FUNCTION_BLOCK PUBLIC FB_LogToDisk // Regularly writes contents of the log to disk
// Once the log file reaches a set size, a new log file is created.
// If the max number of files is reached, the oldest file is discarded.
VAR CONSTANT
	MAX_ITEMS_IN_BUFFER : UDINT := 20; // Should be long enough to allow for worst case writes (where an old file has to be deleted and a new file created).  
	CRLF : STRING := '$R$L'; // Windows style line ending
END_VAR
VAR_INPUT
	bEnable : BOOL; // If enabled, log items will be written to disk
END_VAR
VAR_OUTPUT
	bFault 				: BOOL; // An error occured while trying to add to log or write to disk
	sFaultDescription	: STRING[80]; // Detailed error information
	bLoggerInitialized  : BOOL; // True the first time the logger has ran through all states (ie., after succesfully writing the first log message and emptying the buffer)
	sCurrentLogFile		: T_MaxString; // The file which is currently used for logging (and can be viewed for instance by the HMI)
END_VAR
VAR
	// Properties set by FB_init
	sLogFolder 			: T_MaxString;
	sLogFilePrefix 		: T_MaxString;
	sLogFileExtension 	: T_MaxString;
	nMaxLogFileSize 	: ULINT; // [bytes] When this size is reached, a new log file is created 
	nMaxNumberOfLogFiles: UINT;

	// State machine
	fbStateMachine 	: FB_StateMachine;	
	eState 			: E_LogToDiskState := E_LogToDiskState.InitializeFBs;
	
	// Log item buffer
	stLogItemFromBuffer : UDT_LogItem; // Log item retrieved from the buffer	
	stLogItemToDisk		: UDT_LogItem; // Log item to be written to the log file
	cbBuffer 	: ARRAY[1..(MAX_ITEMS_IN_BUFFER * (SIZEOF(UDT_LogItem) + 4))] OF BYTE; // Note that the buffer size is larger than the number of items * item size, because 4 bytes are added to each item by FB_MemRingBuffer
	fbBuffer 	: FB_MemRingBuffer := (pBuffer:= ADR(cbBuffer), cbBuffer:= SIZEOF(cbBuffer));

	// File function blocks (asynchronous)
	fbFileOpen			: FB_FileOpen; // https://infosys.beckhoff.com/content/1033/tcplclib_tc2_system/30977547.html
	fbFilePuts			: FB_FilePuts; // https://infosys.beckhoff.com/content/1033/tcplclib_tc2_system/30979083.html
	fbFileClose			: FB_FileClose; // https://infosys.beckhoff.com/content/1033/tcplclib_tc2_system/30972939.html
	fbFileProperties	: FB_FileProperties; // https://infosys.beckhoff.com/content/1033/tcplclib_tc2_utilities/10047843595.html
    fbEnumFiles			: FB_EnumFindFileEntry; // https://infosys.beckhoff.com/content/1033/tcplclib_tc2_utilities/34982539.html
	fbFileDelete		: FB_FileDelete; // https://infosys.beckhoff.com/content/1033/tcplclib_tc2_system/30974475.html

	sPath: STRING; // Path to the current log file
	
	tOldestLogFile 	: ST_FindFileEntry; // Reference to the oldest log file in the log folder
	nFileCount		: UINT; // Number of log files found  
	
	fbFormatString : FB_FormatString; // https://infosys.beckhoff.com/content/1033/tcplclib_tc2_utilities/34990219.html
END_VAR
VAR_TEMP
	fMonth : REAL;
	fDay : REAL;
	fHour : REAL;
	fMinute : REAL;
	fSecond : REAL;
	fMilliseconds : REAL;
	sLevel : T_MaxString;

	nFileSize : ULINT;
	
	stEmptyLogItem : UDT_LogItem;
END_VAR

fbStateMachine(nState := eState);

CASE eState OF
	E_LogToDiskState.InitializeFBs:
		// Initialize function blocks
		fbFileOpen(
			bExecute := FALSE,
			ePath := PATH_GENERIC,
		);
		fbFilePuts(bExecute := FALSE);
		fbFileClose(bExecute := FALSE);
		fbFileProperties(bExecute := FALSE);
		fbEnumFiles(bExecute := FALSE);
		fbFileDelete(
			bExecute := FALSE,
			ePath := PATH_GENERIC,
		);
		
		eState := E_LogToDiskState.WaitForCommand;

	E_LogToDiskState.WaitForCommand:
		IF bEnable THEN
			IF (stLogItemFromBuffer.sMsg = '') THEN
				stLogItemFromBuffer := Pop();
			ELSE
				eState := E_LogToDiskState.OpenOrCreateFile;
			END_IF
		END_IF

	E_LogToDiskState.OpenOrCreateFile:
		IF fbStateMachine.bStateChanged THEN
			// Create a new file path if none was given (i.e., after reboot or when file size limit has been reached)
			IF (sPath = '') THEN
				sPath := CreatePath();
			END_IF  	
		END_IF
		fbFileOpen(
			bExecute := TRUE,	
			sPathName := sPath, 
			nMode := FOPEN_MODEAPPEND OR FOPEN_MODETEXT, // Open file in read/write text mode
		);
		IF (NOT fbFileOpen.bBusy) THEN
			fbFileOpen(bExecute := FALSE);
			IF fbFileOpen.bError THEN
				fbFormatString(sFormat := 'Unable to open file (error code 0x%X)', arg1 := F_UDINT(fbFileOpen.nErrId), sOut => sFaultDescription);
				eState := E_LogToDiskState.Error;
			ELSE
				sCurrentLogFile := sPath;
				eState := E_LogToDiskState.CheckFileSize;
			END_IF
		END_IF

	E_LogToDiskState.CheckFileSize:
		fbFileProperties(
			bExecute := TRUE,	
			sPathName := sPath 
		);
		IF (NOT fbFileProperties.bBusy) THEN
			fbFileProperties(bExecute := FALSE);
			IF fbFileProperties.bError THEN
				fbFormatString(sFormat := 'Unable to get file properties (error code 0x%X)', arg1 := F_UDINT(fbFileProperties.nErrId), sOut => sFaultDescription);
				eState := E_LogToDiskState.Error;
			ELSE
				// Check file size
				// ST_FindFileEntry info at https://infosys.beckhoff.com/content/1033/tcplclib_tc2_utilities/35363851.html
				nFileSize := ULARGE_TO_ULINT(fbFileProperties.stProperties.fileSize);
				IF (nFileSize >= nMaxLogFileSize) THEN
					// Create a final log item for this log file
					stLogItemToDisk.eLevel := E_LogLevel.DEBUG;
					fbFormatString(
						sFormat := 'File size exceeded (%u/%u bytes), creating new file.',
						arg1 := F_ULINT(nFileSize),
						arg2 := F_ULINT(nMaxLogFileSize),
						sOut => stLogItemToDisk.sMsg
					);
					stLogItemToDisk.stTimestamp := Sys_Variables.SystemTime_TS;
					sPath := ''; // Trigger new file creation
				ELSE
					stLogItemToDisk := stLogItemFromBuffer; // Set log item to be written to disk
					stLogItemFromBuffer := stEmptyLogItem; // Clear log item from buffer to trigger new item pop
				END_IF
				eState := E_LogToDiskState.WriteLogItemPrefix;
			END_IF
		END_IF
	
	E_LogToDiskState.WriteLogItemPrefix:
		IF fbStateMachine.bStateChanged THEN
			// Build a prefix string, e.g. '[2022-02-04 12:13:45.343] INFO; '

			// Suppress error "VAR_IN_OUT parameter 'in' needs variable with write access as input."	
			fMonth := WORD_TO_REAL(stLogItemToDisk.stTimestamp.wMonth); 
			fDay := WORD_TO_REAL(stLogItemToDisk.stTimestamp.wDay); 
			fHour := WORD_TO_REAL(stLogItemToDisk.stTimestamp.wHour); 
			fMinute := WORD_TO_REAL(stLogItemToDisk.stTimestamp.wMinute); 
			fSecond := WORD_TO_REAL(stLogItemToDisk.stTimestamp.wSecond); 
			fMilliseconds := WORD_TO_REAL(stLogItemToDisk.stTimestamp.wMilliseconds);
			sLevel := TO_STRING(stLogItemToDisk.eLevel);
 
			fbFormatString(
				sFormat := '[%u-%02.0f-%02.0f %02.0f:%02.0f:%02.0f.%03.0f] %s: ',
				arg1 := F_WORD(stLogItemToDisk.stTimestamp.wYear),
				arg2 := F_REAL(fMonth),
				arg3 := F_REAL(fDay),
				arg4 := F_REAL(fHour),
				arg5 := F_REAL(fMinute),
				arg6 := F_REAL(fSecond),
				arg7 := F_REAL(fMilliseconds),
				arg8 := F_STRING(sLevel),
				sOut => fbFilePuts.sLine
			);
		END_IF
		fbFilePuts(bExecute := TRUE, hFile := fbFileOpen.hFile);
		IF (NOT fbFilePuts.bBusy) THEN
			fbFilePuts(bExecute := FALSE);
			IF fbFilePuts.bError THEN
				fbFormatString(sFormat := 'Unable to write log record to file (error code 0x%X)', arg1 := F_UDINT(fbFilePuts.nErrId), sOut => sFaultDescription);
				eState := E_LogToDiskState.Error;
			ELSE // Done, write the log message
				eState := E_LogToDiskState.WriteLogItemMessage;
			END_IF
		END_IF
	
	E_LogToDiskState.WriteLogItemMessage:
		IF fbStateMachine.bStateChanged THEN
			fbFilePuts.sLine := CONCAT(stLogItemToDisk.sMsg, CRLF); 	
		END_IF
		fbFilePuts(bExecute := TRUE, hFile := fbFileOpen.hFile);
		IF (NOT fbFilePuts.bBusy) THEN
			fbFilePuts(bExecute := FALSE);
			IF fbFilePuts.bError THEN
				fbFormatString(sFormat := 'Unable to write log record to file (error code 0x%X)', arg1 := F_UDINT(fbFilePuts.nErrId), sOut => sFaultDescription);
				eState := E_LogToDiskState.Error;
			ELSE // Done, get the next log item in the buffer
				IF (stLogItemFromBuffer.sMsg <> '') THEN 
					// Last log item retrieved from the buffer wasn't written yet (e.g., after new file creation), so no need to pop items from the buffer yet
					eState := E_LogToDiskState.CloseFile;
				ELSE // Check if there are more items in the buffer
					stLogItemFromBuffer := Pop();
					IF (stLogItemFromBuffer.sMsg = '') THEN // Buffer empty, close the file
						eState := E_LogToDiskState.CloseFile;
					ELSE // More items to be written, but first check file size before adding more items
						eState := E_LogToDiskState.CheckFileSize;
					END_IF
				END_IF
			END_IF
		END_IF
	
	E_LogToDiskState.CloseFile:
		fbFileClose(bExecute := TRUE, hFile := fbFileOpen.hFile);
		IF (NOT fbFileClose.bBusy) THEN
			fbFileClose(bExecute := FALSE);
			IF fbFileClose.bError THEN
				fbFormatString(sFormat := 'Unable to close file (error code 0x%X)', arg1 := F_UDINT(fbFileClose.nErrId), sOut => sFaultDescription);
				eState := E_LogToDiskState.Error;
			ELSE
				eState := E_LogToDiskState.FindObsoleteFiles;
			END_IF
		END_IF
	
	E_LogToDiskState.FindObsoleteFiles:
		// Delete oldest log files in log folder until we're at MAX_NUMBER_OF_LOG_FILES
		IF fbStateMachine.bStateChanged THEN
			nFileCount := 0;	
			tOldestLogFile.sFileName := ''; 
			// Create a path search string, e.g. '/tmp/Log_*.txt'
			fbFormatString(
				sFormat := '%s/%s*.%s',
				arg1 := F_STRING(sLogFolder),
				arg2 := F_STRING(sLogFilePrefix),
				arg3 := F_STRING(sLogFileExtension),
				sOut => fbEnumFiles.sPathName
			);
			fbEnumFiles.eCmd := E_EnumCmdType.eEnumCmd_First;
		END_IF
		fbEnumFiles(bExecute := TRUE);
		IF (NOT fbEnumFiles.bBusy) THEN
			fbEnumFiles(bExecute := FALSE, eCmd := E_EnumCmdType.eEnumCmd_Next);
			IF fbEnumFiles.bError THEN
				fbFormatString(
					sFormat := 'Unable to get files in folder "%s" (error code 0x%X)',
					arg1 := F_STRING(fbEnumFiles.sPathName),
					arg2 := F_UDINT(fbEnumFiles.nErrId),
					sOut => sFaultDescription
				);
				eState := E_LogToDiskState.Error;
			ELSIF fbEnumFiles.bEOE THEN
				// Found all files, carry on
				eState := E_LogToDiskState.WaitForCommand;
				bLoggerInitialized := TRUE;
			ELSE
				// Found a file, check if it's older than the previous find
				nFileCount := nFileCount + 1;
				IF (tOldestLogFile.sFileName = '') 
					OR (PLWORD_TO_LWORD(ADR(fbEnumFiles.stFindFile.creationTime)) < PLWORD_TO_LWORD(ADR(tOldestLogFile.creationTime))) 
				THEN
					tOldestLogFile := fbEnumFiles.stFindFile;
				END_IF
				IF (nFileCount > nMaxNumberOfLogFiles) THEN
					// Max number of log files reached, delete the file				
					eState := E_LogToDiskState.DeleteFile;
				END_IF
			END_IF
		END_IF

	E_LogToDiskState.DeleteFile:
		IF fbStateMachine.bStateChanged THEN
			fbFormatString(
				sFormat := '%s/%s',
				arg1 := F_STRING(sLogFolder),
				arg2 := F_STRING(tOldestLogFile.sFileName),
				sOut => fbFileDelete.sPathName
			);
		END_IF
		fbFileDelete(bExecute := TRUE);
		IF (NOT fbFileDelete.bBusy) THEN
			fbFileDelete(bExecute := FALSE);
			IF fbFileDelete.bError THEN
				fbFormatString(
					sFormat := 'Unable to delete file "%s" (error code 0x%X)',
					arg1 := F_STRING(tOldestLogFile.sFileName),
					arg2 := F_UDINT(fbFileClose.nErrId), 
					sOut => sFaultDescription
				);
				eState := E_LogToDiskState.Error;
			ELSE // Done deleting, continue searching for obsolete files
				eState := E_LogToDiskState.FindObsoleteFiles;
			END_IF
		END_IF

	E_LogToDiskState.Error:
		IF (sFaultDescription = '') THEN
			sFaultDescription := 'Unknown error';
		END_IF

END_CASE

bFault S= (eState = E_LogToDiskState.Error);

METHOD PROTECTED AddToLog
VAR_INPUT
	sMsg : T_MaxString; // The message to be logged
	eLevel : E_LogLevel; // Log level (debug, info, warn, etc.)
END_VAR
VAR
	bOk : BOOL;
	stLogItem : UDT_LogItem;
	nMaxItems : UDINT;
END_VAR
// Ignore empty messages or messages when the logger has an error
IF (sMsg = '') OR bFault THEN
	RETURN;
END_IF

stLogItem.sMsg := sMsg;
stLogItem.eLevel := eLevel;
stLogItem.stTimestamp := Sys_Variables.SystemTime_TS;

fbBuffer.A_AddTail(
	pWrite := ADR(stLogItem),
	cbWrite := SIZEOF(stLogItem),
	bOk => bOk,
);

IF NOT bOk THEN // Buffer overflow
	// Make sure no more items will be added to the log
	bFault := TRUE;
	// Pop last item to make room for the famous last words
	Pop(); 
	// And add those words to the log
	nMaxItems := MAX_ITEMS_IN_BUFFER;
	fbFormatString(
		sFormat := 'Log buffer size limit (%u) reached! Dumping buffer and disabling the logger.',
		arg1 := F_UDINT(nMaxItems),
		sOut => sFaultDescription
	);
	stLogItem.sMsg := sFaultDescription;
	stLogItem.eLevel := E_LogLevel.FATAL;
	fbBuffer.A_AddTail(
		pWrite := ADR(stLogItem),
		cbWrite := SIZEOF(stLogItem),
		bOk => bOk,
	);
END_IF
END_METHOD

METHOD PROTECTED CreatePath : STRING // Create a filename with a date/time stamp, e.g. "/tmp/Log_20230203-093610.txt'
VAR
	fMonth : REAL;
	fDay : REAL;
	fHour : REAL;
	fMinute : REAL;
	fSecond : REAL;
END_VAR
{warning 'TODO: test on windows platform'}

// Suppress error "VAR_IN_OUT parameter 'in' needs variable with write access as input."	
fMonth := WORD_TO_REAL(Sys_Variables.SystemTime_TS.wMonth); 
fDay := WORD_TO_REAL(Sys_Variables.SystemTime_TS.wDay); 
fHour := WORD_TO_REAL(Sys_Variables.SystemTime_TS.wHour); 
fMinute := WORD_TO_REAL(Sys_Variables.SystemTime_TS.wMinute); 
fSecond := WORD_TO_REAL(Sys_Variables.SystemTime_TS.wSecond); 

fbFormatString(
	sFormat := '%s/%s%u%02.0f%02.0f-%02.0f%02.0f%02.0f.%s',
	arg1 := F_STRING(sLogFolder),
	arg2 := F_STRING(sLogFilePrefix),
	arg3 := F_WORD(Sys_Variables.SystemTime_TS.wYear),
	arg4 := F_REAL(fMonth),
	arg5 := F_REAL(fDay),
	arg6 := F_REAL(fHour),
	arg7 := F_REAL(fMinute),
	arg8 := F_REAL(fSecond),
	arg9 := F_STRING(sLogFileExtension),
	sOut => CreatePath
);
END_METHOD

METHOD PUBLIC DEBUG // Add a message to the log with log level DEBUG 
(*
The DEBUG level is used for logging messages that help developers find out what went wrong
during a debugging session. While the specifics of what messages to log at the DEBUG level
is dependent on your application, you generally want to include detailed information that
can help developers troubleshoot an issue quickly. 
This can include variable state in the surrounding scope, or relevant error codes.
Unlike TRACE, DEBUG level logging can be turned on in production without making the application unusable,
but it should not be left on indefinitely to ensure the log is not flooded.
*)
VAR_INPUT
	sMsg : T_MaxString; // The message to be logged
END_VAR
THIS^.AddToLog(sMsg, E_LogLevel.DEBUG);
END_METHOD

METHOD PUBLIC ERROR // Add a message to the log with log level ERROR
(*
The ERROR log level is used to represent error conditions in a system that
prevent a specific operation from running, but the system itself can continue
working even if it is at a reduced level of functionality or performance.
Generally, ERROR logs should be investigated as soon as possible but they don't
carry the same urgency as FATAL messages since the system can continue working.
*)
VAR_INPUT
	sMsg : T_MaxString; // The message to be logged
END_VAR
THIS^.AddToLog(sMsg, E_LogLevel.ERROR);
END_METHOD

METHOD PUBLIC FATAL // Add a message to the log with log level FATAL
(*
The FATAL log level annotates messages with the greatest severity.
It usually means that something critical is broken, and the system cannot continue to do any more
useful work without the intervention of an engineer. T
ypically, such entries are logged before the system is shut down ("famous last words").
*)
VAR_INPUT
	sMsg : T_MaxString; // The message to be logged
END_VAR
THIS^.AddToLog(sMsg, E_LogLevel.FATAL);
END_METHOD

METHOD FB_init : BOOL
VAR_INPUT
	bInitRetains : BOOL; // if TRUE, the retain variables are initialized (warm start / cold start)
	bInCopyCode : BOOL;  // if TRUE, the instance afterwards gets moved into the copy code (online change)

	sLogFolder 			: T_MaxString; // Example for TwinCAT/BSD: '/tmp'. The folder where log files will be stored. Do not add trailing '/' or '\'. 
	sLogFilePrefix 		: T_MaxString; // Example: 'Log_'
	sLogFileExtension 	: T_MaxString; // Example: 'txt'
	nMaxLogFileSize 	: ULINT; // [bytes] When this size is reached, a new log file is created 
	nMaxNumberOfLogFiles: UINT;
END_VAR
THIS^.sLogFolder := sLogFolder;
THIS^.sLogFilePrefix := sLogFilePrefix;
THIS^.sLogFileExtension := sLogFileExtension;
THIS^.nMaxLogFileSize := nMaxLogFileSize;
THIS^.nMaxNumberOfLogFiles := nMaxNumberOfLogFiles;
END_METHOD

METHOD PUBLIC INFO // Add a message to the log with log level INFO
(*
INFO-level messages indicate events in the system that are significant to the
general purpose of the system. Such events are logged to show that the system is
operating normally. For example, a recipe was started or stopped. 
Production systems typically default to logging at this level so that a 
summary of the application's normal behavior is visible to anyone reading the logs.
*)
VAR_INPUT
	sMsg : T_MaxString; // The message to be logged
END_VAR
THIS^.AddToLog(sMsg, E_LogLevel.INFO);
END_METHOD

METHOD PROTECTED Pop : UDT_LogItem; // Pops the buffer head (returns the oldest log item in the buffer)
fbBuffer.A_RemoveHead(
	pRead:= ADR(Pop),
	cbRead:= SIZEOF(Pop),
);
END_METHOD

METHOD PUBLIC TRACE // Add a message to the log with log level TRACE
(*
The TRACE level can be used for tracing the path of code execution in a program.
Generally, TRACE is used for showing the flow of the program, and to provide a detailed breakdown of the sequence
of events that led to a crash, a silent failure, an error, or some other event logged at a different level.
The TRACE level is only used temporarily (when the code is a "work in progress").
*)
VAR_INPUT
	sMsg : T_MaxString; // The message to be logged
END_VAR
THIS^.AddToLog(sMsg, E_LogLevel.TRACE);
END_METHOD

METHOD PUBLIC WARN // Add a message to the log with log level WARN
(*
Messages logged at the WARN level typically indicate that something unexpected happened,
but the system can recover and continue to function normally.
It is mainly used to draw attention to situations that should be addressed soon before
they pose a problem for the system.
*)
VAR_INPUT
	sMsg : T_MaxString; // The message to be logged
END_VAR
THIS^.AddToLog(sMsg, E_LogLevel.WARN);
END_METHOD

END_FUNCTION_BLOCK

(* stored: Version 1.1.0.1, ProductVersion 3.1.4024.11
   POU FB_LogToDisk: Id {a722563c-1b3c-082f-3710-fb1c23b337b0}, SpecialFunc None
   Folder Private: Id {06ea4b8b-8b88-05b4-114a-e159875a95a0}
   Folder Public: Id {690da83f-5550-0084-3e92-f3004d90cd65}
   Method AddToLog: Id {bff9ee33-3717-027a-138b-f9964612e88c}
   Method CreatePath: Id {28455913-5a7f-004f-3c48-f7a0c0ab7d6c}
   Method DEBUG: Id {73f740e6-2a7d-0335-2d60-04f04456d0fa}
   Method ERROR: Id {56e0a7f0-dba1-0134-25e6-42b1ca5ad6dd}
   Method FATAL: Id {9dea5fac-8f6f-00f5-025c-86cdbbb5c16f}
   Method FB_init: Id {3e31473c-86c3-0ff7-324f-81de8ebfd10c}
   Method INFO: Id {129ab2a5-c74e-0bad-1ca8-3aaada834c1f}
   Method Pop: Id {d6331dd4-6e1f-043e-18b0-d56bd8407d9a}
   Method TRACE: Id {852b99e3-4aae-02e1-20be-be286b738a87}
   Method WARN: Id {6d9befb4-3cad-0f4d-268e-38de03686e94} *)
